FUNCTION_BLOCK ResetTask EXTENDS TcoCore.TcoTask IMPLEMENTS ITcoDriveSimple
VAR
    {attribute 'hide'}
    _axisRef : REFERENCE TO TcoAxisRef;
    {attribute 'hide'}
    _mcReset : Tc2_MC2.MC_Reset;
END_VAR

IF NOT __ISVALIDREF(_axisRef) THEN
    IF __ISVALIDREF(DriveRef) THEN
        _axisRef REF= DriveRef.AxisRef;
    ELSE
        RETURN;
    END_IF
END_IF

IF Execute() THEN
    _mcReset(Axis := _axisRef);

    DoneWhen(_mcReset.Done);
    ThrowWhen(_mcReset.Error);
END_IF

PROPERTY DriveRef : REFERENCE TO TcoDriveSimple
GET
VAR
    _drive : ITcoDriveSimple := 0;
END_VAR
IF __QUERYINTERFACE(THIS^.Parent, _drive) THEN
    DriveRef REF= _drive.DriveRef;
END_IF
END_GET
END_PROPERTY

METHOD PUBLIC FB_init : BOOL
VAR_INPUT
    bInitRetains : BOOL; // if TRUE, the retain variables are initialized (warm start / cold start)
    bInCopyCode : BOOL; // if TRUE, the instance afterwards gets moved into the copy code (online change)
  	ParentObject : ITcoObject;	
END_VAR
SUPER^.FB_init(bInitRetains := bInitRetains, bInCopyCode := bInCopyCode, ParentObject := ParentObject);
END_METHOD

(*~
	<docu>
		<summary>
			Executes when task reaches the ```Done``` state .
		</summary>			
	</docu>	
~*)
METHOD PROTECTED OnDone
DriveRef.RestoreTasks();
DriveRef.ClearError();

_mcReset(Axis := _axisRef,Execute := FALSE);
END_METHOD

(*~
	<docu>
		<summary>
			Executes when task reaches the ```Error``` state.
			<para>
				Do not confuse with <see cref="PlcDocu.TcoCore.TcoTask.WhileError()"/>, that is called cyclically until '''Error''' state is left.
			</para>
		</summary>			
	</docu>	
~*)
METHOD PROTECTED OnError
DriveRef.RestoreTasks();

IF NOT _axisRef.Status.Error THEN
    DriveRef.SetErrorID(DriveRef._resetTask._mcReset.ErrorID);
END_IF

_mcReset(Axis := _axisRef, Execute := FALSE);
END_METHOD

METHOD PROTECTED OnStart
DriveRef.ClearError();

_mcReset(Axis := _axisRef,Execute := TRUE);
END_METHOD

(*~
	<docu>
		<summary>
			Restores this instance to the Ready state. Can be called explicitly or from within one of the restore mechanisms.
			<para>
				See also <see cref="PlcDocu.TcoCore.TcoTask.AutoRestorable()"/>
			</para>
		</summary>			
	</docu>	
~*)
METHOD Restore : ITcoRestorable
SUPER^.Restore();
END_METHOD

(*~
	<docu>
		<summary>
			Executes until task is in ```Error``` state .
		</summary>			
	</docu>	
~*)
METHOD PROTECTED WhileError
IF NOT _axisRef.Status.Error THEN
	DriveRef.SetErrorID(DriveRef._resetTask._mcReset.ErrorID);
    _mcReset(Axis := _axisRef, Execute := FALSE);	
END_IF
END_METHOD

END_FUNCTION_BLOCK

(* stored: Version 1.1.0.1, ProductVersion 3.1.4024.9
   POU ResetTask: Id {018ad7d5-79df-023a-3c91-a698bbbc60f2}, SpecialFunc None
   Property DriveRef: Id {539bbd16-3d54-0366-3b1b-e22e7261b0a1}
   Get Get: Id {16dc8c5c-3663-033c-27c5-32406243dfc0}
   Method FB_init: Id {6855e6dd-82b3-081c-24eb-2aeb53c9e8eb}
   Method OnDone: Id {72d4d2a3-5082-0045-31b5-fff519bd5b2b}
   Method OnError: Id {317d0d1d-7213-0f6a-002c-bd29fc6a14f6}
   Method OnStart: Id {2c8c79ff-94f6-08a3-2eaa-65d37d102a58}
   Method Restore: Id {b66f0f12-7e1b-0ae5-3d39-d75ff6b45738}
   Method WhileError: Id {70772925-0ea5-0b7e-21de-df87b76e125e} *)
